// SIMATIC S7-200 project (STEP 7-Micro/WIN), CPU 224 REL 02.01

SYMBOL_TABLE USUARIO1
P_PARO           I0.0
P_MARCHA         I0.1
FC_C_LLENO       I0.2
FC_C_REPOSO      I0.3
FC_C_VOLCADO     I0.4
FC_IZQUIERDA     I0.5
FC_DERECHA       I0.6
CINTA_1          Q0.0
TRITURADOR       Q0.1
CINTA_2          Q0.2
M3_RECOGIDA_CONTENEDOR Q0.3
M3_VOLCADO_CONTENEDOR Q0.4
M4_IZQUIERDA     Q0.5
M4_DERECHA       Q0.6
END_SYMBOL_TABLE

ORGANIZATION_BLOCK PRINCIPAL:OB1
TITLE=COMENTARIOS DEL PROGRAMA
BEGIN
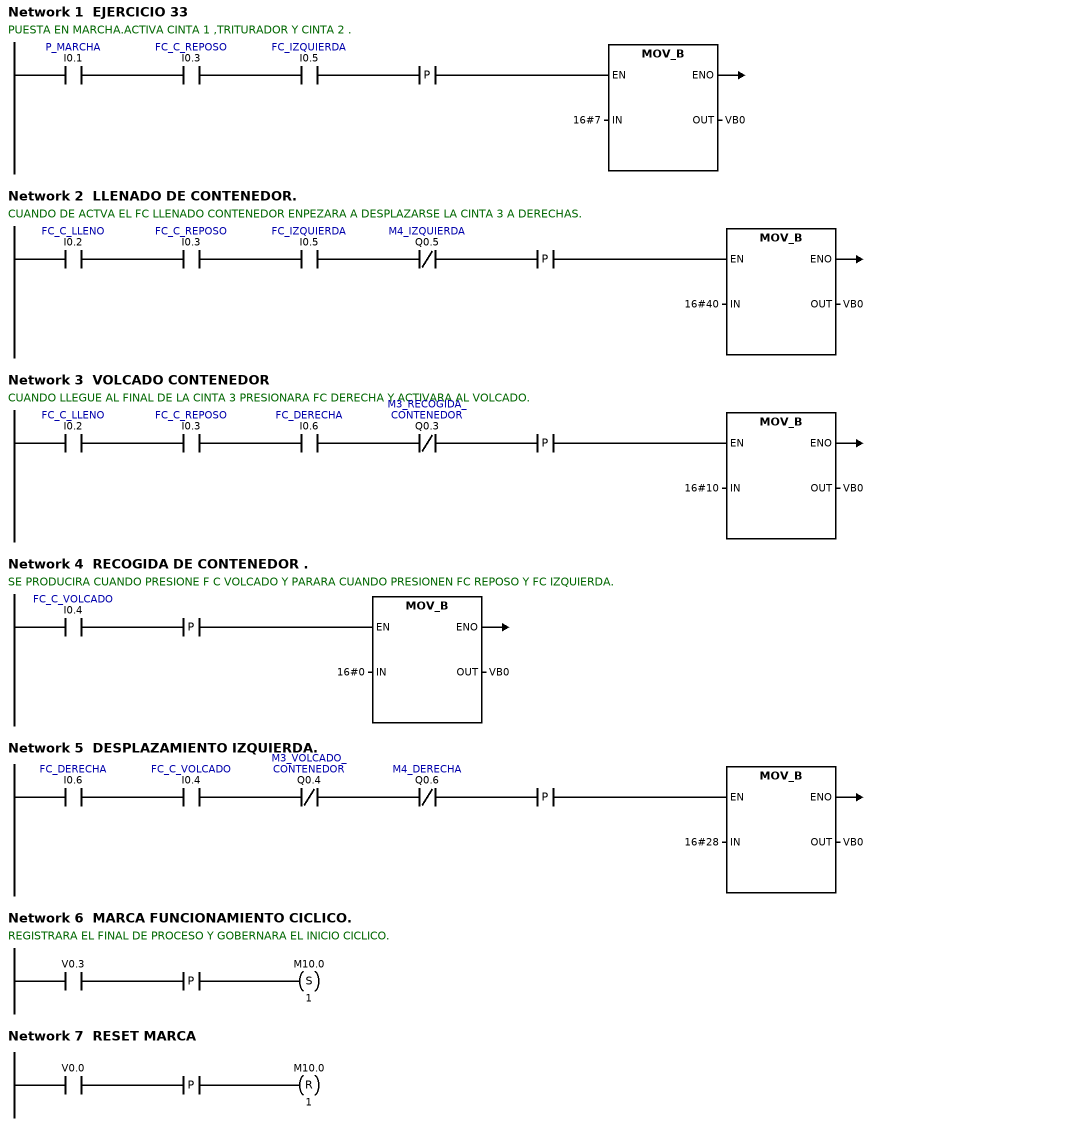
Network 1 // EJERCICIO 33 
// PUESTA EN MARCHA.ACTIVA CINTA 1 ,TRITURADOR Y CINTA 2 .
LD     P_MARCHA:I0.1
A      FC_C_REPOSO:I0.3
A      FC_IZQUIERDA:I0.5
EU
MOVB   16#7, VB0
Network 2 // LLENADO DE CONTENEDOR.
// CUANDO DE ACTVA EL FC LLENADO CONTENEDOR ENPEZARA A DESPLAZARSE LA CINTA 3 A DERECHAS.
LD     FC_C_LLENO:I0.2
A      FC_C_REPOSO:I0.3
A      FC_IZQUIERDA:I0.5
AN     M4_IZQUIERDA:Q0.5
EU
MOVB   16#40, VB0
Network 3 // VOLCADO CONTENEDOR
// CUANDO LLEGUE AL FINAL DE LA CINTA 3 PRESIONARA FC DERECHA Y ACTIVARA AL VOLCADO.
LD     FC_C_LLENO:I0.2
A      FC_C_REPOSO:I0.3
A      FC_DERECHA:I0.6
AN     M3_RECOGIDA_CONTENEDOR:Q0.3
EU
MOVB   16#10, VB0
Network 4 // RECOGIDA DE CONTENEDOR .
// SE PRODUCIRA CUANDO PRESIONE F C VOLCADO Y PARARA CUANDO PRESIONEN FC REPOSO Y FC IZQUIERDA.
LD     FC_C_VOLCADO:I0.4
EU
MOVB   16#0, VB0
Network 5 // DESPLAZAMIENTO IZQUIERDA.
LD     FC_DERECHA:I0.6
A      FC_C_VOLCADO:I0.4
AN     M3_VOLCADO_CONTENEDOR:Q0.4
AN     M4_DERECHA:Q0.6
EU
MOVB   16#28, VB0
Network 6 // MARCA FUNCIONAMIENTO CICLICO.
// REGISTRARA EL FINAL DE PROCESO Y GOBERNARA EL INICIO CICLICO.
LD     V0.3
EU
S      M10.0, 1
Network 7 // RESET MARCA 
LD     V0.0
EU
R      M10.0, 1
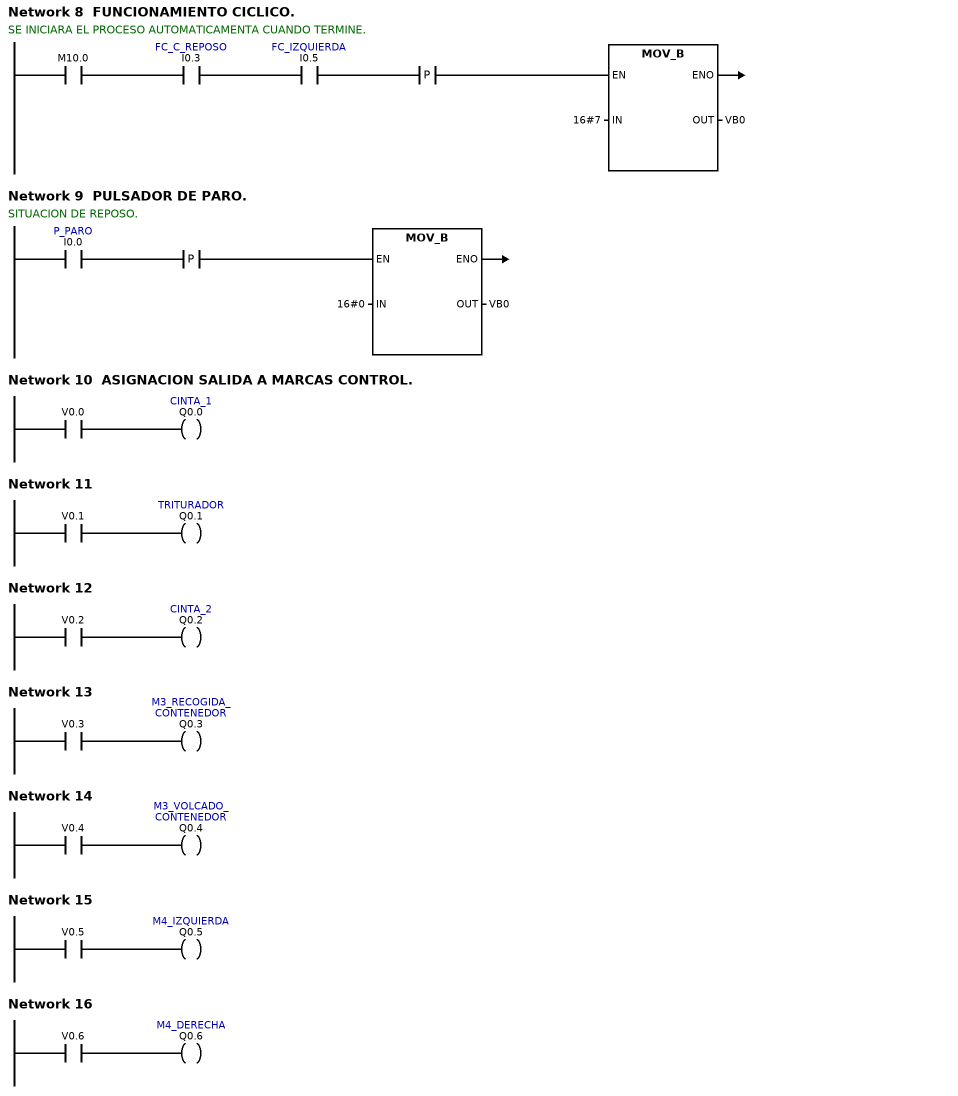
Network 8 // FUNCIONAMIENTO CICLICO.
// SE INICIARA EL PROCESO AUTOMATICAMENTA CUANDO TERMINE.
LD     M10.0
A      FC_C_REPOSO:I0.3
A      FC_IZQUIERDA:I0.5
EU
MOVB   16#7, VB0
Network 9 // PULSADOR DE PARO.
// SITUACION DE REPOSO.
LD     P_PARO:I0.0
EU
MOVB   16#0, VB0
Network 10 // ASIGNACION SALIDA A MARCAS CONTROL.
LD     V0.0
=      CINTA_1:Q0.0
Network 11
LD     V0.1
=      TRITURADOR:Q0.1
Network 12
LD     V0.2
=      CINTA_2:Q0.2
Network 13
LD     V0.3
=      M3_RECOGIDA_CONTENEDOR:Q0.3
Network 14
LD     V0.4
=      M3_VOLCADO_CONTENEDOR:Q0.4
Network 15
LD     V0.5
=      M4_IZQUIERDA:Q0.5
Network 16
LD     V0.6
=      M4_DERECHA:Q0.6
END_ORGANIZATION_BLOCK
